FUNCTION_BLOCK AR2IO_TO_AR (* Composite FB for convert AR2IO to AR *)
  (* Standard: 61499-2; Description: Copyright (c) 2024 HR Agrartechnik GmbH This program and the accompanying materials are made available under the terms of the Eclipse Public License 2.0 which is available at https://www.eclipse.org/legal/epl-2.0/ SPDX-License-Identifier: EPL-2.0 *)
  (* Version 1.0, 2024-04-24, Franz Höpfinger, HR Agrartechnik GmbH *)
  PACKAGE adapter::conversion::bidirectional;
  IMPORT eclipse4diac::core::TypeHash;
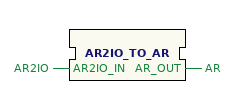
  SOCKETS
    AR2IO_IN : adapter::types::bidirectional::AR2IO(D1 := 0.0); (* AR2IO Adapter Input *)
  END_SOCKETS
  PLUGS
    AR_OUT : adapter::types::unidirectional::AR; (* AR Adapter Output *)
  END_PLUGS
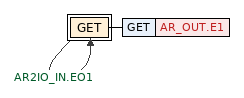
  EC_STATES
    GET : GET -> AR_OUT.E1;
  END_STATES
  EC_TRANSITIONS
    GET TO GET := AR2IO_IN.EO1;
  END_TRANSITIONS
  ALGORITHM GET IN ST:
AR_OUT.D1 := AR2IO_IN.D1;
  END_ALGORITHM
END_FUNCTION_BLOCK
